// TIA Portal V20 export
FUNCTION_BLOCK "LER_AxisControl_InterlockSummary"   // FB230, LAD
// stored: Access Published, MemoryReserve 100, SetENOAutomatically false
   VAR_INPUT
      enableManualCmds : Bool;
      interlockSource { ExternalAccessible := 'False'; ExternalVisible := 'False'; ExternalWritable := 'False'} : "typeAxisInterlockSource";
   END_VAR
   VAR_OUTPUT
      interlockcGeneral : Bool;
   END_VAR
   VAR_IN_OUT
      moduleInterface : "LBC_typeAxisControlInterface";
      controlNode : "LBC_typeAxisControlNode";
   END_VAR
   VAR
      statProcessValuesCommands { S7_SetPoint := 'True'} : "LBC_typeAxisControlNodeCommands";
      statAnyInterlockAlive { S7_SetPoint := 'True'} : Bool;
   END_VAR
   VAR CONSTANT
      TRUE : Bool := TRUE;
      FALSE : Bool := FALSE;
   END_VAR
BEGIN

REGION Network 1: Command Capture (HMI / ControlNode arbitration)
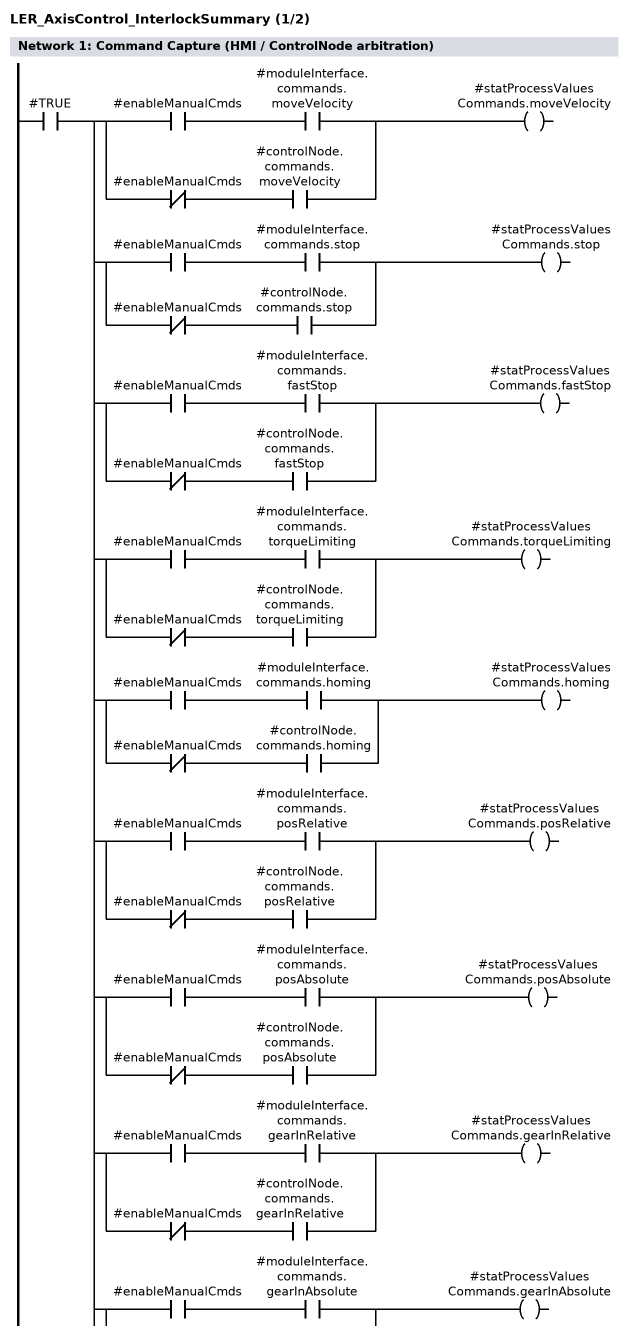
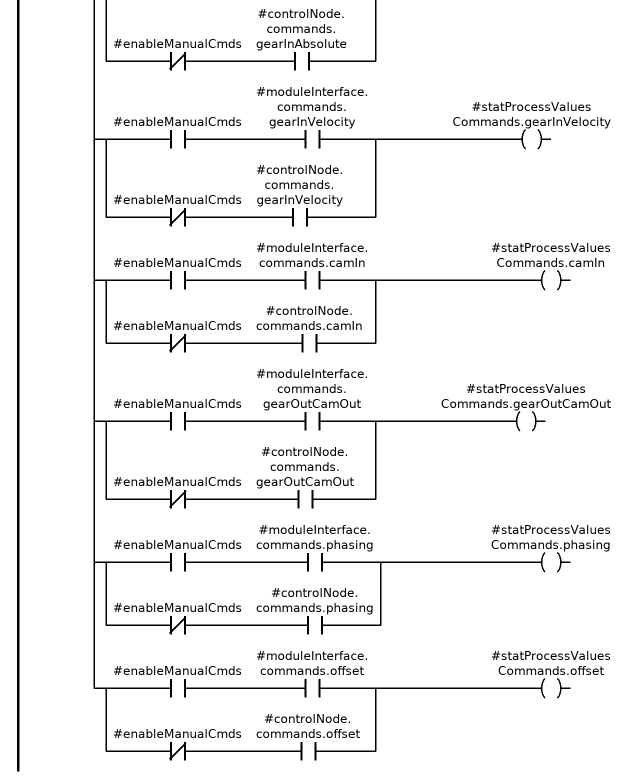
   RUNG wire#powerrail
      Contact( #TRUE )
      wire#w1
      Contact( #enableManualCmds )
      Contact( #moduleInterface.commands.moveVelocity )
      wire#w2
      Coil( #statProcessValuesCommands.moveVelocity )
   END_RUNG
   RUNG wire#w1
      I_Contact( #enableManualCmds )
      Contact( #controlNode.commands.moveVelocity )
   END_RUNG wire#w2
   RUNG wire#w1
      Contact( #enableManualCmds )
      Contact( #moduleInterface.commands.stop )
      wire#w3
      Coil( #statProcessValuesCommands.stop )
   END_RUNG
   RUNG wire#w1
      I_Contact( #enableManualCmds )
      Contact( #controlNode.commands.stop )
   END_RUNG wire#w3
   RUNG wire#w1
      Contact( #enableManualCmds )
      Contact( #moduleInterface.commands.fastStop )
      wire#w4
      Coil( #statProcessValuesCommands.fastStop )
   END_RUNG
   RUNG wire#w1
      I_Contact( #enableManualCmds )
      Contact( #controlNode.commands.fastStop )
   END_RUNG wire#w4
   RUNG wire#w1
      Contact( #enableManualCmds )
      Contact( #moduleInterface.commands.torqueLimiting )
      wire#w5
      Coil( #statProcessValuesCommands.torqueLimiting )
   END_RUNG
   RUNG wire#w1
      I_Contact( #enableManualCmds )
      Contact( #controlNode.commands.torqueLimiting )
   END_RUNG wire#w5
   RUNG wire#w1
      Contact( #enableManualCmds )
      Contact( #moduleInterface.commands.homing )
      wire#w6
      Coil( #statProcessValuesCommands.homing )
   END_RUNG
   RUNG wire#w1
      I_Contact( #enableManualCmds )
      Contact( #controlNode.commands.homing )
   END_RUNG wire#w6
   RUNG wire#w1
      Contact( #enableManualCmds )
      Contact( #moduleInterface.commands.posRelative )
      wire#w7
      Coil( #statProcessValuesCommands.posRelative )
   END_RUNG
   RUNG wire#w1
      I_Contact( #enableManualCmds )
      Contact( #controlNode.commands.posRelative )
   END_RUNG wire#w7
   RUNG wire#w1
      Contact( #enableManualCmds )
      Contact( #moduleInterface.commands.posAbsolute )
      wire#w8
      Coil( #statProcessValuesCommands.posAbsolute )
   END_RUNG
   RUNG wire#w1
      I_Contact( #enableManualCmds )
      Contact( #controlNode.commands.posAbsolute )
   END_RUNG wire#w8
   RUNG wire#w1
      Contact( #enableManualCmds )
      Contact( #moduleInterface.commands.gearInRelative )
      wire#w9
      Coil( #statProcessValuesCommands.gearInRelative )
   END_RUNG
   RUNG wire#w1
      I_Contact( #enableManualCmds )
      Contact( #controlNode.commands.gearInRelative )
   END_RUNG wire#w9
   RUNG wire#w1
      Contact( #enableManualCmds )
      Contact( #moduleInterface.commands.gearInAbsolute )
      wire#w10
      Coil( #statProcessValuesCommands.gearInAbsolute )
   END_RUNG
   RUNG wire#w1
      I_Contact( #enableManualCmds )
      Contact( #controlNode.commands.gearInAbsolute )
   END_RUNG wire#w10
   RUNG wire#w1
      Contact( #enableManualCmds )
      Contact( #moduleInterface.commands.gearInVelocity )
      wire#w11
      Coil( #statProcessValuesCommands.gearInVelocity )
   END_RUNG
   RUNG wire#w1
      I_Contact( #enableManualCmds )
      Contact( #controlNode.commands.gearInVelocity )
   END_RUNG wire#w11
   RUNG wire#w1
      Contact( #enableManualCmds )
      Contact( #moduleInterface.commands.camIn )
      wire#w12
      Coil( #statProcessValuesCommands.camIn )
   END_RUNG
   RUNG wire#w1
      I_Contact( #enableManualCmds )
      Contact( #controlNode.commands.camIn )
   END_RUNG wire#w12
   RUNG wire#w1
      Contact( #enableManualCmds )
      Contact( #moduleInterface.commands.gearOutCamOut )
      wire#w13
      Coil( #statProcessValuesCommands.gearOutCamOut )
   END_RUNG
   RUNG wire#w1
      I_Contact( #enableManualCmds )
      Contact( #controlNode.commands.gearOutCamOut )
   END_RUNG wire#w13
   RUNG wire#w1
      Contact( #enableManualCmds )
      Contact( #moduleInterface.commands.phasing )
      wire#w14
      Coil( #statProcessValuesCommands.phasing )
   END_RUNG
   RUNG wire#w1
      I_Contact( #enableManualCmds )
      Contact( #controlNode.commands.phasing )
   END_RUNG wire#w14
   RUNG wire#w1
      Contact( #enableManualCmds )
      Contact( #moduleInterface.commands.offset )
      wire#w15
      Coil( #statProcessValuesCommands.offset )
   END_RUNG
   RUNG wire#w1
      I_Contact( #enableManualCmds )
      Contact( #controlNode.commands.offset )
   END_RUNG wire#w15
   // the same network as SCL:
   #statProcessValuesCommands.moveVelocity := #TRUE AND ((#enableManualCmds AND #moduleInterface.commands.moveVelocity) OR (NOT #enableManualCmds AND #controlNode.commands.moveVelocity));
   #statProcessValuesCommands.stop := #TRUE AND ((#enableManualCmds AND #moduleInterface.commands.stop) OR (NOT #enableManualCmds AND #controlNode.commands.stop));
   #statProcessValuesCommands.fastStop := #TRUE AND ((#enableManualCmds AND #moduleInterface.commands.fastStop) OR (NOT #enableManualCmds AND #controlNode.commands.fastStop));
   #statProcessValuesCommands.torqueLimiting := #TRUE AND ((#enableManualCmds AND #moduleInterface.commands.torqueLimiting) OR (NOT #enableManualCmds AND #controlNode.commands.torqueLimiting));
   #statProcessValuesCommands.homing := #TRUE AND ((#enableManualCmds AND #moduleInterface.commands.homing) OR (NOT #enableManualCmds AND #controlNode.commands.homing));
   #statProcessValuesCommands.posRelative := #TRUE AND ((#enableManualCmds AND #moduleInterface.commands.posRelative) OR (NOT #enableManualCmds AND #controlNode.commands.posRelative));
   #statProcessValuesCommands.posAbsolute := #TRUE AND ((#enableManualCmds AND #moduleInterface.commands.posAbsolute) OR (NOT #enableManualCmds AND #controlNode.commands.posAbsolute));
   #statProcessValuesCommands.gearInRelative := #TRUE AND ((#enableManualCmds AND #moduleInterface.commands.gearInRelative) OR (NOT #enableManualCmds AND #controlNode.commands.gearInRelative));
   #statProcessValuesCommands.gearInAbsolute := #TRUE AND ((#enableManualCmds AND #moduleInterface.commands.gearInAbsolute) OR (NOT #enableManualCmds AND #controlNode.commands.gearInAbsolute));
   #statProcessValuesCommands.gearInVelocity := #TRUE AND ((#enableManualCmds AND #moduleInterface.commands.gearInVelocity) OR (NOT #enableManualCmds AND #controlNode.commands.gearInVelocity));
   #statProcessValuesCommands.camIn := #TRUE AND ((#enableManualCmds AND #moduleInterface.commands.camIn) OR (NOT #enableManualCmds AND #controlNode.commands.camIn));
   #statProcessValuesCommands.gearOutCamOut := #TRUE AND ((#enableManualCmds AND #moduleInterface.commands.gearOutCamOut) OR (NOT #enableManualCmds AND #controlNode.commands.gearOutCamOut));
   #statProcessValuesCommands.phasing := #TRUE AND ((#enableManualCmds AND #moduleInterface.commands.phasing) OR (NOT #enableManualCmds AND #controlNode.commands.phasing));
   #statProcessValuesCommands.offset := #TRUE AND ((#enableManualCmds AND #moduleInterface.commands.offset) OR (NOT #enableManualCmds AND #controlNode.commands.offset));
END_REGION

REGION Network 2: Interlock State Matrix (Which Interlocks Are Active)
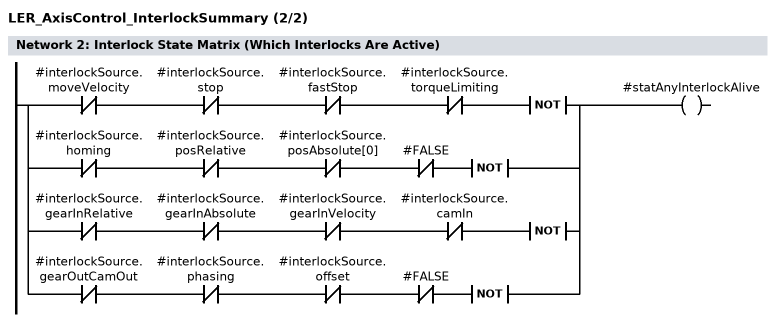
   RUNG wire#powerrail
      I_Contact( #interlockSource.moveVelocity )
      I_Contact( #interlockSource.stop )
      I_Contact( #interlockSource.fastStop )
      I_Contact( #interlockSource.torqueLimiting )
      Not()
      wire#w1
      Coil( #statAnyInterlockAlive )
   END_RUNG
   RUNG wire#powerrail
      I_Contact( #interlockSource.homing )
      I_Contact( #interlockSource.posRelative )
      I_Contact( #interlockSource.posAbsolute[0] )
      I_Contact( #FALSE )
      Not()
   END_RUNG wire#w1
   RUNG wire#powerrail
      I_Contact( #interlockSource.gearInRelative )
      I_Contact( #interlockSource.gearInAbsolute )
      I_Contact( #interlockSource.gearInVelocity )
      I_Contact( #interlockSource.camIn )
      Not()
   END_RUNG wire#w1
   RUNG wire#powerrail
      I_Contact( #interlockSource.gearOutCamOut )
      I_Contact( #interlockSource.phasing )
      I_Contact( #interlockSource.offset )
      I_Contact( #FALSE )
      Not()
   END_RUNG wire#w1
   // the same network as SCL:
   #statAnyInterlockAlive := NOT (NOT #interlockSource.moveVelocity AND NOT #interlockSource.stop AND NOT #interlockSource.fastStop AND NOT #interlockSource.torqueLimiting) OR NOT (NOT #interlockSource.homing AND NOT #interlockSource.posRelative AND NOT #interlockSource.posAbsolute[0] AND NOT #FALSE) OR NOT (NOT #interlockSource.gearInRelative AND NOT #interlockSource.gearInAbsolute AND NOT #interlockSource.gearInVelocity AND NOT #interlockSource.camIn) OR NOT (NOT #interlockSource.gearOutCamOut AND NOT #interlockSource.phasing AND NOT #interlockSource.offset AND NOT #FALSE);
END_REGION

REGION Network 3 (SCL): Active Motion Interlock Arbitration
   IF #statProcessValuesCommands.moveVelocity OR (#controlNode.monitoring.moveVelocitySelected AND #controlNode.monitoring.commandBusy) THEN
       #interlockcGeneral := #interlockSource.moveVelocity;

   ELSIF #statProcessValuesCommands.stop AND (#controlNode.monitoring.stopSelected AND #controlNode.monitoring.commandDone) THEN
       #interlockcGeneral := #interlockSource.stop;

   ELSIF #statProcessValuesCommands.fastStop AND (#controlNode.monitoring.fastStopSelected AND #controlNode.monitoring.commandDone) THEN
       #interlockcGeneral := #interlockSource.fastStop;

   ELSIF #statProcessValuesCommands.torqueLimiting OR (#controlNode.monitoring.torqueLimitingSelected AND #controlNode.monitoring.commandBusy) THEN
       #interlockcGeneral := #interlockSource.torqueLimiting;

   ELSIF #statProcessValuesCommands.homing OR (#controlNode.monitoring.homingSelected AND #controlNode.monitoring.commandBusy) THEN
       #interlockcGeneral := #interlockSource.homing;

   ELSIF #statProcessValuesCommands.posRelative OR (#controlNode.monitoring.posRelativeSelected AND #controlNode.monitoring.commandBusy) THEN
       #interlockcGeneral := #interlockSource.posRelative;

   ELSIF #statProcessValuesCommands.posAbsolute OR (#controlNode.monitoring.posAbsoluteSelected AND #controlNode.monitoring.commandBusy) THEN
       #interlockcGeneral := #interlockSource.posAbsolute[0];

   ELSIF #statProcessValuesCommands.gearInRelative OR (#controlNode.monitoring.gearInRelativeSelected AND #controlNode.monitoring.commandBusy) THEN
       #interlockcGeneral := #interlockSource.gearInRelative;

   ELSIF #statProcessValuesCommands.gearInAbsolute AND (#controlNode.monitoring.gearInAbsoluteSelected AND #controlNode.monitoring.commandBusy) THEN
       #interlockcGeneral := #interlockSource.gearInAbsolute;

   ELSIF #statProcessValuesCommands.gearInVelocity AND (#controlNode.monitoring.gearInVelocitySelected AND #controlNode.monitoring.commandBusy) THEN
       #interlockcGeneral := #interlockSource.gearInVelocity;

   ELSIF #statProcessValuesCommands.camIn AND (#controlNode.monitoring.camInSelected AND #controlNode.monitoring.commandBusy) THEN
       #interlockcGeneral := #interlockSource.camIn;

   ELSIF #statProcessValuesCommands.gearOutCamOut AND (#statProcessValuesCommands.gearOutCamOut AND #controlNode.monitoring.commandDone) OR #controlNode.monitoring.inSync THEN
       #interlockcGeneral := #interlockSource.gearInVelocity;

   ELSIF #statProcessValuesCommands.phasing AND (#controlNode.monitoring.phasingSelected AND #controlNode.monitoring.commandBusy) THEN
       #interlockcGeneral := #interlockSource.phasing;

   ELSIF #statProcessValuesCommands.offset AND (#controlNode.monitoring.offsetSelected AND #controlNode.monitoring.commandBusy) THEN
       #interlockcGeneral := #interlockSource.offset;

   ELSE
       #interlockcGeneral := #statAnyInterlockAlive;
   END_IF;
END_REGION
END_FUNCTION_BLOCK
